// TIA Portal V17 export
// export: Created 2023-02-13T11:16:47.3031872Z, ExportSetting WithDefaults, DisplayName Totally Integrated Automation Portal, DisplayVersion V17, DisplayName TIA Portal Openness, DisplayVersion V17, DisplayName TIA Portal Teamcenter Gateway, DisplayVersion V17, DisplayName TIA Portal Version Control Interface, DisplayVersion V17, DisplayName SINAMICS Startdrive Advanced, DisplayVersion V17, DisplayName SINAMICS Startdrive G130, G150, S120, S150, SINAMICS MV, S210, DisplayVersion V17, DisplayName SINAMICS Startdrive G110M, G120, G120C, G120D, G120P, G115D, DisplayVersion V17, DisplayName STEP 7 Professional, DisplayVersion V17, DisplayName STEP 7 Safety, DisplayVersion V17, DisplayName WinCC Professional, DisplayVersion V17
FUNCTION "Transfer_Homomix" : Void   // FC9, LAD
{ S7_Optimized_Access := 'TRUE' }
VERSION : 0.1
// stored: AutoNumber true, IsIECCheckEnabled false, SetENOAutomatically false, UDAEnableTagReadback false
   VAR_INPUT
      req : Bool;
      "low level" : Bool;
      "tank inload" : Bool;
      "cmd start" : Bool;
      "cmd stop" : Bool;
      "FB AV Transfer" : Bool;
      "FB SV Pump" : Bool;
   END_VAR
   VAR_OUTPUT
      "AV Transfer" : Bool;
      "SV Pump" : Bool;
      indicator_start : Bool;
      indicator_stop : Bool;
   END_VAR
   VAR_IN_OUT
      "cmd en start" : Bool;
      "cmd en stop" : Bool;
      "cmd state start" : Bool;
      "cmd state stop" : Bool;
      indicator_request : Bool;
      "always ON" : Bool;
   END_VAR
   VAR_TEMP   // added for the SCL form of the ladder/FBD networks
      _w1 : Bool;
      _w2 : Bool;
   END_VAR
BEGIN

REGION Network 1
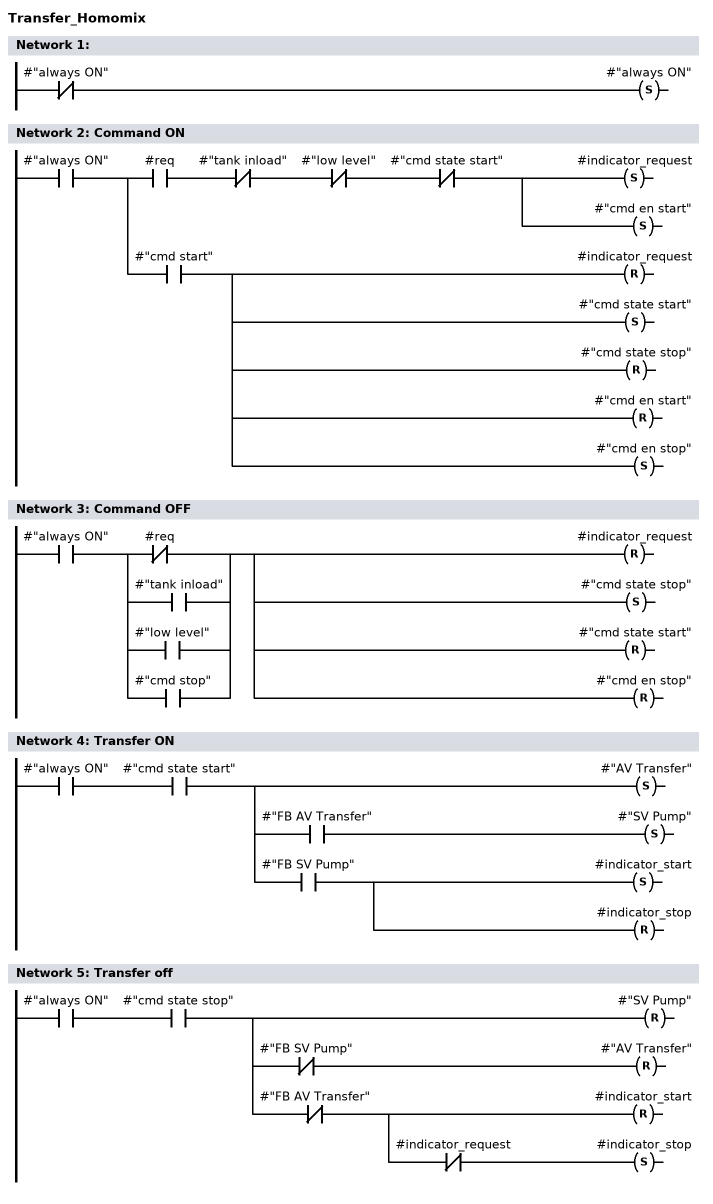
   RUNG wire#powerrail
      I_Contact( #"always ON" )
      S_Coil( #"always ON" )
   END_RUNG
   // the same network as SCL:
   IF NOT #"always ON" THEN #"always ON" := TRUE; END_IF;
END_REGION

REGION Network 2: Command ON
   RUNG wire#powerrail
      Contact( #"always ON" )
      wire#w1
      Contact( #req )
      I_Contact( #"tank inload" )
      I_Contact( #"low level" )
      I_Contact( #"cmd state start" )
      wire#w2
      S_Coil( #indicator_request )
   END_RUNG
   RUNG wire#w2
      S_Coil( #"cmd en start" )
   END_RUNG
   RUNG wire#w1
      Contact( #"cmd start" )
      wire#w3
      R_Coil( #indicator_request )
   END_RUNG
   RUNG wire#w3
      S_Coil( #"cmd state start" )
   END_RUNG
   RUNG wire#w3
      R_Coil( #"cmd state stop" )
   END_RUNG
   RUNG wire#w3
      R_Coil( #"cmd en start" )
   END_RUNG
   RUNG wire#w3
      S_Coil( #"cmd en stop" )
   END_RUNG
   // the same network as SCL:
   IF #"always ON" AND #req AND NOT #"tank inload" AND NOT #"low level" AND NOT #"cmd state start" THEN
       #indicator_request := TRUE;
       #"cmd en start" := TRUE;
   END_IF;
   IF #"always ON" AND #"cmd start" THEN
       #indicator_request := FALSE;
       #"cmd state start" := TRUE;
       #"cmd state stop" := FALSE;
       #"cmd en start" := FALSE;
       #"cmd en stop" := TRUE;
   END_IF;
END_REGION

REGION Network 3: Command OFF
   RUNG wire#powerrail
      Contact( #"always ON" )
      wire#w1
      I_Contact( #req )
      wire#w2
      R_Coil( #indicator_request )
   END_RUNG
   RUNG wire#w1
      Contact( #"tank inload" )
   END_RUNG wire#w2
   RUNG wire#w1
      Contact( #"low level" )
   END_RUNG wire#w2
   RUNG wire#w1
      Contact( #"cmd stop" )
   END_RUNG wire#w2
   RUNG wire#w2
      S_Coil( #"cmd state stop" )
   END_RUNG
   RUNG wire#w2
      R_Coil( #"cmd state start" )
   END_RUNG
   RUNG wire#w2
      R_Coil( #"cmd en stop" )
   END_RUNG
   // the same network as SCL:
   IF #"always ON" AND (NOT #req OR #"tank inload" OR #"low level" OR #"cmd stop") THEN
       #indicator_request := FALSE;
       #"cmd state stop" := TRUE;
       #"cmd state start" := FALSE;
       #"cmd en stop" := FALSE;
   END_IF;
END_REGION

REGION Network 4: Transfer ON
   RUNG wire#powerrail
      Contact( #"always ON" )
      Contact( #"cmd state start" )
      wire#w1
      S_Coil( #"AV Transfer" )
   END_RUNG
   RUNG wire#w1
      Contact( #"FB AV Transfer" )
      S_Coil( #"SV Pump" )
   END_RUNG
   RUNG wire#w1
      Contact( #"FB SV Pump" )
      wire#w2
      S_Coil( #indicator_start )
   END_RUNG
   RUNG wire#w2
      R_Coil( #indicator_stop )
   END_RUNG
   // the same network as SCL:
   #_w1 := #"always ON" AND #"cmd state start";
   IF #_w1 THEN #"AV Transfer" := TRUE; END_IF;
   IF #_w1 AND #"FB AV Transfer" THEN #"SV Pump" := TRUE; END_IF;
   IF #_w1 AND #"FB SV Pump" THEN
       #indicator_start := TRUE;
       #indicator_stop := FALSE;
   END_IF;
END_REGION

REGION Network 5: Transfer off
   RUNG wire#powerrail
      Contact( #"always ON" )
      Contact( #"cmd state stop" )
      wire#w1
      R_Coil( #"SV Pump" )
   END_RUNG
   RUNG wire#w1
      I_Contact( #"FB SV Pump" )
      R_Coil( #"AV Transfer" )
   END_RUNG
   RUNG wire#w1
      I_Contact( #"FB AV Transfer" )
      wire#w2
      R_Coil( #indicator_start )
   END_RUNG
   RUNG wire#w2
      I_Contact( #indicator_request )
      S_Coil( #indicator_stop )
   END_RUNG
   // the same network as SCL:
   #_w1 := #"always ON" AND #"cmd state stop";
   IF #_w1 THEN #"SV Pump" := FALSE; END_IF;
   IF #_w1 AND NOT #"FB SV Pump" THEN #"AV Transfer" := FALSE; END_IF;
   #_w2 := #_w1 AND NOT #"FB AV Transfer";
   IF #_w2 THEN #indicator_start := FALSE; END_IF;
   IF #_w2 AND NOT #indicator_request THEN #indicator_stop := TRUE; END_IF;
END_REGION
END_FUNCTION
